(* PLC project SafeLOGIC-1, BrAutomation SafeDESIGNER  4.3.4.4 *)
(* stored: companyURL http://www.br-automation.com, creationDateTime Thu Dec 17 12:56:32 2020 *)

PROGRAM Main

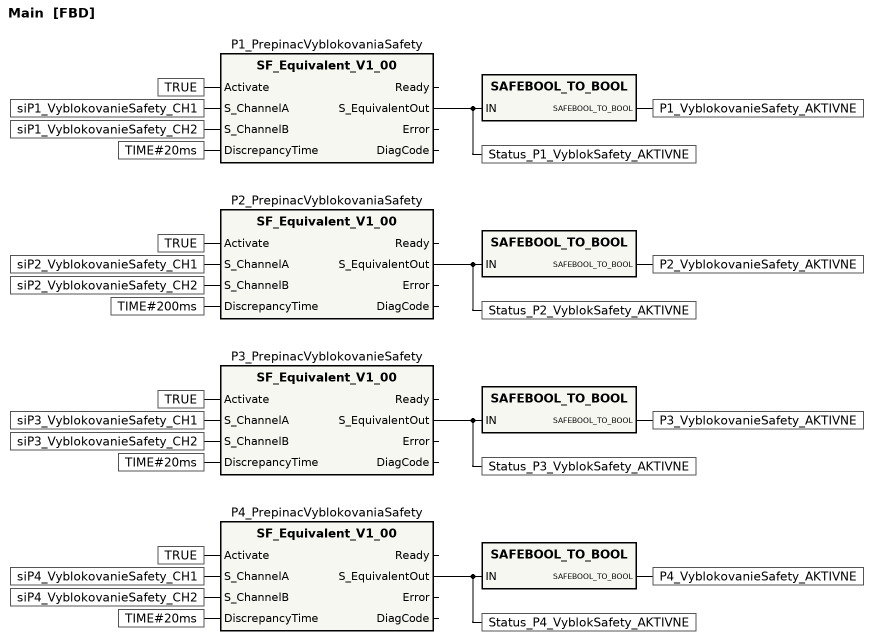
(* FBD diagram, written out as Structured Text *)
P1_PrepinacVyblokovaniaSafety(Activate := TRUE, S_ChannelA := siP1_VyblokovanieSafety_CH1, S_ChannelB := siP1_VyblokovanieSafety_CH2, DiscrepancyTime := TIME#20ms);
Status_P1_VyblokSafety_AKTIVNE := P1_PrepinacVyblokovaniaSafety.S_EquivalentOut;
P1_VyblokovanieSafety_AKTIVNE := SAFEBOOL_TO_BOOL(P1_PrepinacVyblokovaniaSafety.S_EquivalentOut);
P2_PrepinacVyblokovaniaSafety(Activate := TRUE, S_ChannelA := siP2_VyblokovanieSafety_CH1, S_ChannelB := siP2_VyblokovanieSafety_CH2, DiscrepancyTime := TIME#200ms);
Status_P2_VyblokSafety_AKTIVNE := P2_PrepinacVyblokovaniaSafety.S_EquivalentOut;
P2_VyblokovanieSafety_AKTIVNE := SAFEBOOL_TO_BOOL(P2_PrepinacVyblokovaniaSafety.S_EquivalentOut);
P3_PrepinacVyblokovanieSafety(Activate := TRUE, S_ChannelA := siP3_VyblokovanieSafety_CH1, S_ChannelB := siP3_VyblokovanieSafety_CH2, DiscrepancyTime := TIME#20ms);
Status_P3_VyblokSafety_AKTIVNE := P3_PrepinacVyblokovanieSafety.S_EquivalentOut;
P3_VyblokovanieSafety_AKTIVNE := SAFEBOOL_TO_BOOL(P3_PrepinacVyblokovanieSafety.S_EquivalentOut);
P4_PrepinacVyblokovaniaSafety(Activate := TRUE, S_ChannelA := siP4_VyblokovanieSafety_CH1, S_ChannelB := siP4_VyblokovanieSafety_CH2, DiscrepancyTime := TIME#20ms);
Status_P4_VyblokSafety_AKTIVNE := P4_PrepinacVyblokovaniaSafety.S_EquivalentOut;
P4_VyblokovanieSafety_AKTIVNE := SAFEBOOL_TO_BOOL(P4_PrepinacVyblokovaniaSafety.S_EquivalentOut);
END_PROGRAM
